{attribute 'GeneratedUsingTerminal: EL5101-0011-0016'}
{attribute addProperty BoxType "EL5101-0011-0016"}
{attribute addProperty Id "Set_counterBOOL1"}
{attribute addProperty CRC "3181003151"}
{attribute addProperty Size "1"}
TYPE Control_BD9A418F :
STRUCT
	{attribute addProperty Name "Set_counter"}
	Set_counter : BOOL;
END_STRUCT
END_TYPE

(* stored: Version 1.2.0.0, ProductVersion 3.1.4024.9
   DUT Control_BD9A418F: Id {e5752b2a-34b3-47fa-b80c-fa84e9be037e} *)
